(* Logix 5000 project; controller SX_V040001_C001 vendor 1 type 14 code 77 rev 16.22; software revision 16.04; part 29 of 35 *)
(* tags used below, declared in another part *)
   ALL_KINDS : INT[90];
   DRIVE : INT[32];
   DRIVE_INTERVAL : INT[8];
   EMPTYING : INT[18];
   G_DInput : DINT[3];
   loading : INT[19];
   louvre : INT[11];
   METERING : INT[44];
   NOTDOS : INT[6];
   PARAMETER : INT[501];
   pointer_recipe_line : DINT;
   REC_NR_BCD_REMOTE : INT[5];
   REC_NR_BCD_STRING : SINT[2];
   RECIPE_GENERAL : INT[405];
   RM_CMD : INT[9];
   TEMP : INT[14];
(* MainProgram, continued *)

ROUTINE RecipeEnd   (* ladder *)
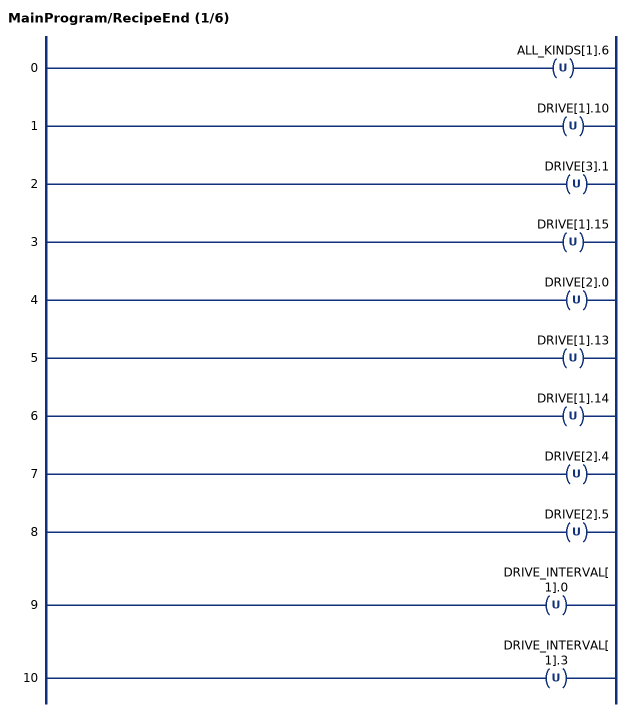
   0: OTU(ALL_KINDS[1].6);
   1: OTU(DRIVE[1].10);
   2: OTU(DRIVE[3].1);
   3: OTU(DRIVE[1].15);
   4: OTU(DRIVE[2].0);
   5: OTU(DRIVE[1].13);
   6: OTU(DRIVE[1].14);
   7: OTU(DRIVE[2].4);
   8: OTU(DRIVE[2].5);
   9: OTU(DRIVE_INTERVAL[1].0);
   10: OTU(DRIVE_INTERVAL[1].3);
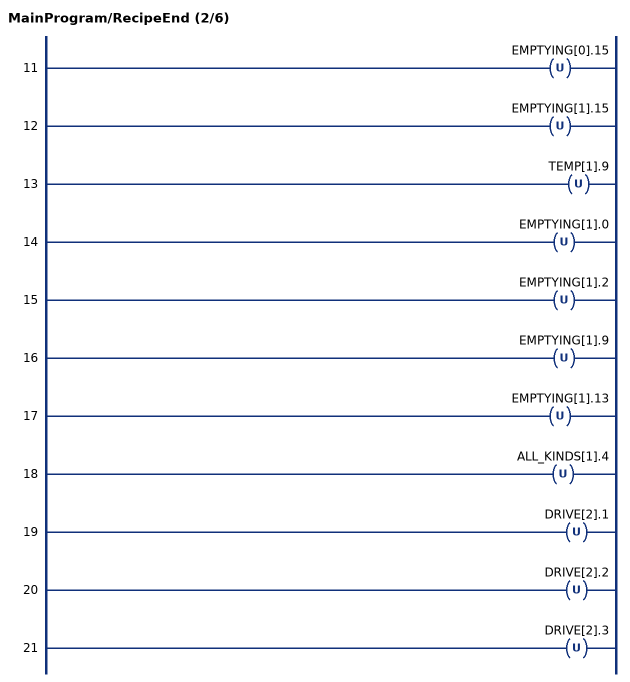
   11: OTU(EMPTYING[0].15);
   12: OTU(EMPTYING[1].15);
   13: OTU(TEMP[1].9);
   14: OTU(EMPTYING[1].0);
   15: OTU(EMPTYING[1].2);
   16: OTU(EMPTYING[1].9);
   17: OTU(EMPTYING[1].13);
   18: OTU(ALL_KINDS[1].4);
   19: OTU(DRIVE[2].1);
   20: OTU(DRIVE[2].2);
   21: OTU(DRIVE[2].3);
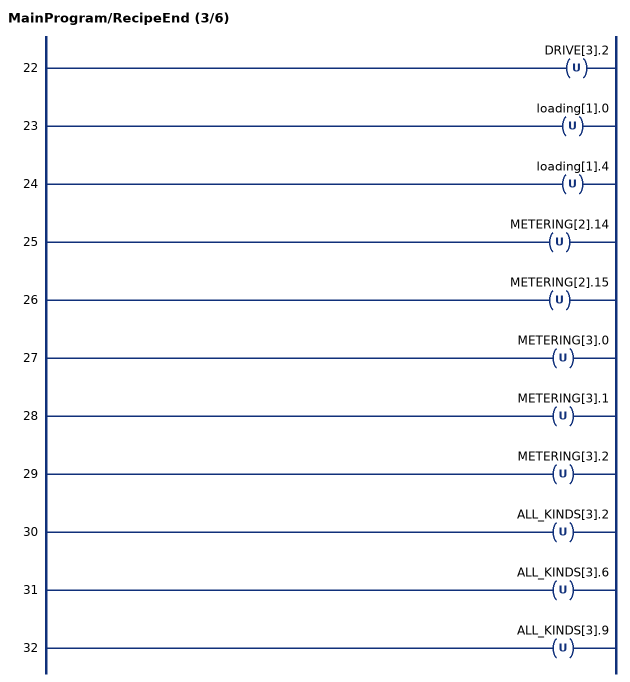
   22: OTU(DRIVE[3].2);
   23: OTU(loading[1].0);
   24: OTU(loading[1].4);
   25: OTU(METERING[2].14);
   26: OTU(METERING[2].15);
   27: OTU(METERING[3].0);
   28: OTU(METERING[3].1);
   29: OTU(METERING[3].2);
   30: OTU(ALL_KINDS[3].2);
   31: OTU(ALL_KINDS[3].6);
   32: OTU(ALL_KINDS[3].9);
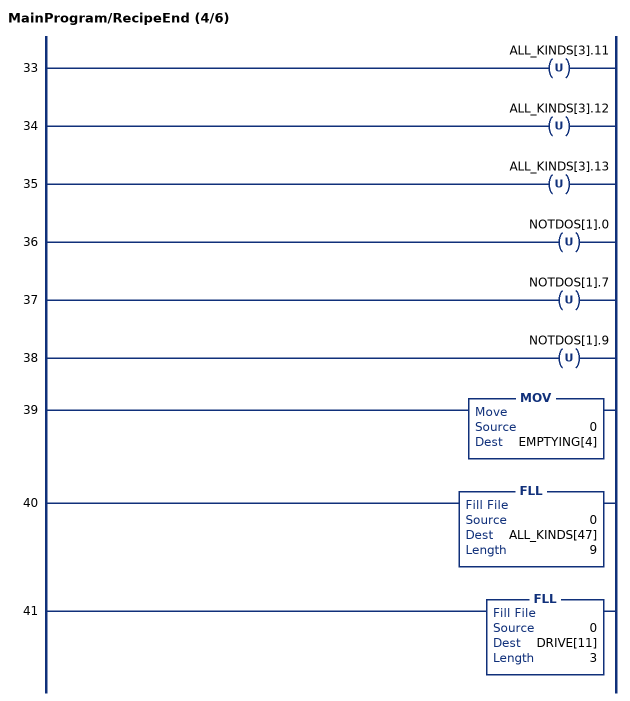
   33: OTU(ALL_KINDS[3].11);
   34: OTU(ALL_KINDS[3].12);
   35: OTU(ALL_KINDS[3].13);
   36: OTU(NOTDOS[1].0);
   37: OTU(NOTDOS[1].7);
   38: OTU(NOTDOS[1].9);
   39: MOV(0,EMPTYING[4]);
   40: FLL(0,ALL_KINDS[47],9);
   41: FLL(0,DRIVE[11],3);
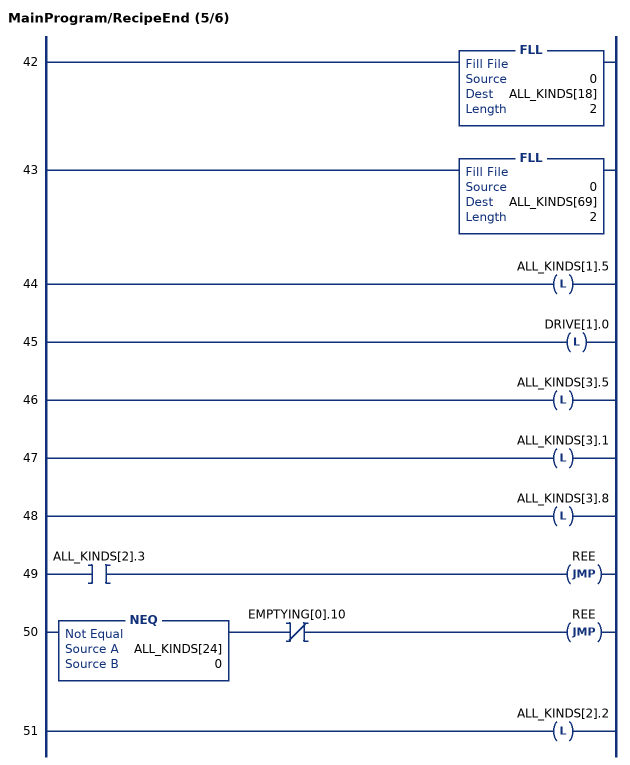
   42: FLL(0,ALL_KINDS[18],2);
   43: FLL(0,ALL_KINDS[69],2);
   44: OTL(ALL_KINDS[1].5);
   45: OTL(DRIVE[1].0);
   46: OTL(ALL_KINDS[3].5);
   47: OTL(ALL_KINDS[3].1);
   48: OTL(ALL_KINDS[3].8);
   49: XIC(ALL_KINDS[2].3)JMP(REE);
   50: NEQ(ALL_KINDS[24],0)XIO(EMPTYING[0].10)JMP(REE);
   51: OTL(ALL_KINDS[2].2);
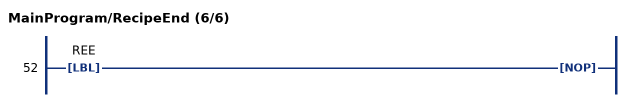
   52: LBL(REE)NOP();
END_ROUTINE

ROUTINE RecipeInterruption   (* ladder *)
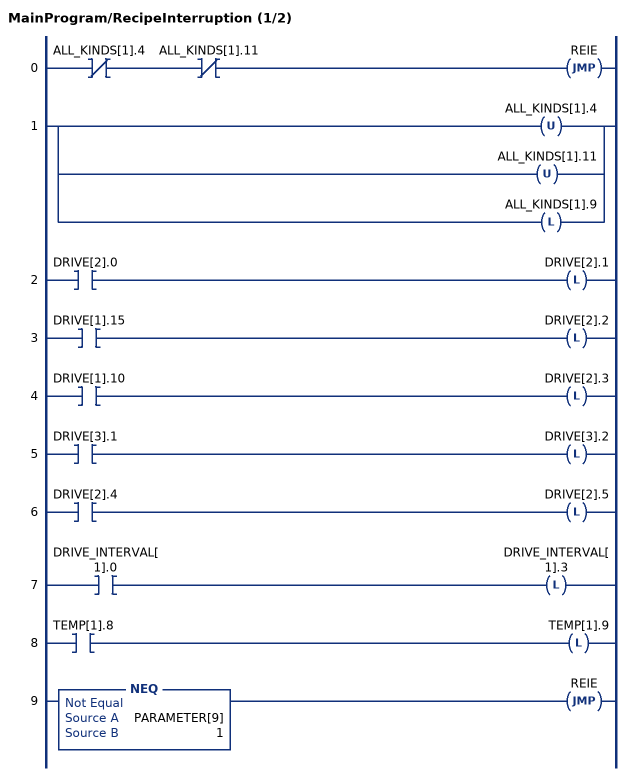
   0: XIO(ALL_KINDS[1].4)XIO(ALL_KINDS[1].11)JMP(REIE);
   1: [OTU(ALL_KINDS[1].4) ,OTU(ALL_KINDS[1].11) ,OTL(ALL_KINDS[1].9) ];
   2: XIC(DRIVE[2].0)OTL(DRIVE[2].1);
   3: XIC(DRIVE[1].15)OTL(DRIVE[2].2);
   4: XIC(DRIVE[1].10)OTL(DRIVE[2].3);
   5: XIC(DRIVE[3].1)OTL(DRIVE[3].2);
   6: XIC(DRIVE[2].4)OTL(DRIVE[2].5);
   7: XIC(DRIVE_INTERVAL[1].0)OTL(DRIVE_INTERVAL[1].3);
   8: XIC(TEMP[1].8)OTL(TEMP[1].9);
   9: NEQ(PARAMETER[9],1)JMP(REIE);
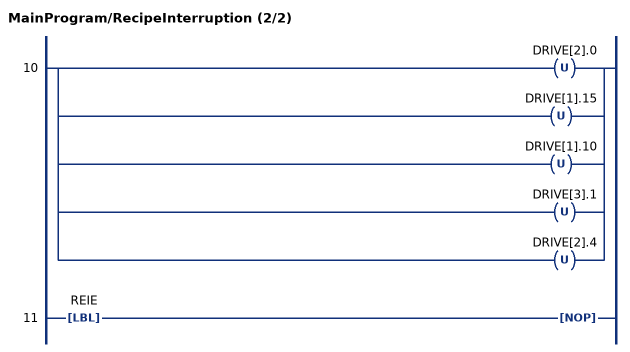
   10: [OTU(DRIVE[2].0) ,OTU(DRIVE[1].15) ,OTU(DRIVE[1].10) ,OTU(DRIVE[3].1) ,OTU(DRIVE[2].4) ];
   11: LBL(REIE)NOP();
END_ROUTINE

ROUTINE RecipeNewstart   (* ladder *)
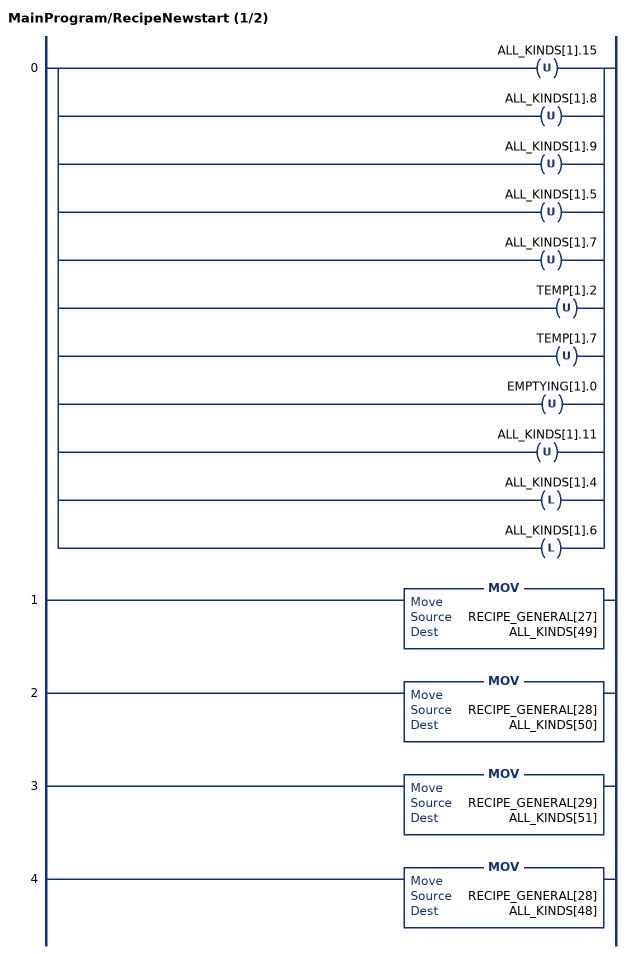
   0: [OTU(ALL_KINDS[1].15) ,OTU(ALL_KINDS[1].8) ,OTU(ALL_KINDS[1].9) ,OTU(ALL_KINDS[1].5) ,OTU(ALL_KINDS[1].7) ,OTU(TEMP[1].2) ,OTU(TEMP[1].7) ,OTU(EMPTYING[1].0) ,OTU(ALL_KINDS[1].11) ,OTL(ALL_KINDS[1].4) ,OTL(ALL_KINDS[1].6) ];
   1: MOV(RECIPE_GENERAL[27],ALL_KINDS[49]);
   2: MOV(RECIPE_GENERAL[28],ALL_KINDS[50]);
   3: MOV(RECIPE_GENERAL[29],ALL_KINDS[51]);
   4: MOV(RECIPE_GENERAL[28],ALL_KINDS[48]);
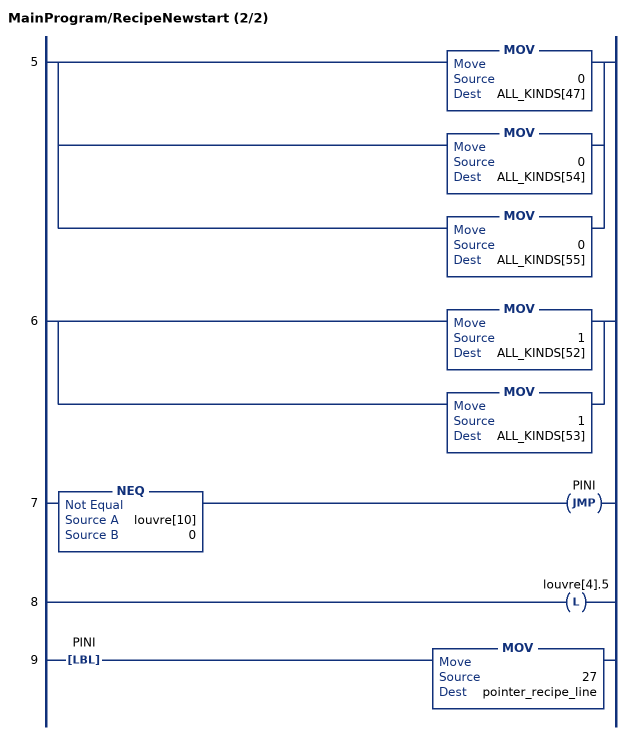
   5: [MOV(0,ALL_KINDS[47]) ,MOV(0,ALL_KINDS[54]) ,MOV(0,ALL_KINDS[55]) ];
   6: [MOV(1,ALL_KINDS[52]) ,MOV(1,ALL_KINDS[53]) ];
   7: NEQ(louvre[10],0)JMP(PINI);
   8: OTL(louvre[4].5);
   9: LBL(PINI)MOV(27,pointer_recipe_line);
END_ROUTINE

ROUTINE RecipeNrBCDin   (* ladder *)
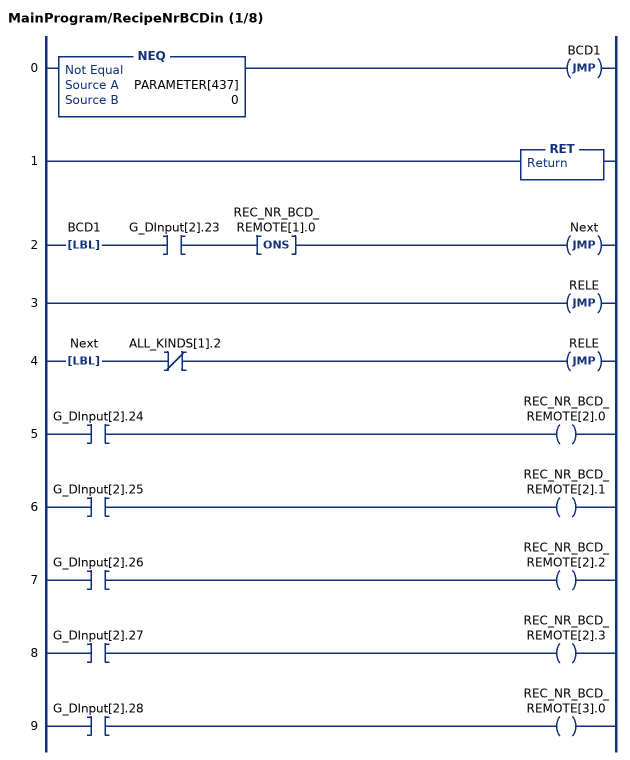
   0: NEQ(PARAMETER[437],0)JMP(BCD1);
   1: RET();
   2: LBL(BCD1)XIC(G_DInput[2].23)ONS(REC_NR_BCD_REMOTE[1].0)JMP(Next);
   3: JMP(RELE);
   4: LBL(Next)XIO(ALL_KINDS[1].2)JMP(RELE);
   5: XIC(G_DInput[2].24)OTE(REC_NR_BCD_REMOTE[2].0);
   6: XIC(G_DInput[2].25)OTE(REC_NR_BCD_REMOTE[2].1);
   7: XIC(G_DInput[2].26)OTE(REC_NR_BCD_REMOTE[2].2);
   8: XIC(G_DInput[2].27)OTE(REC_NR_BCD_REMOTE[2].3);
   9: XIC(G_DInput[2].28)OTE(REC_NR_BCD_REMOTE[3].0);
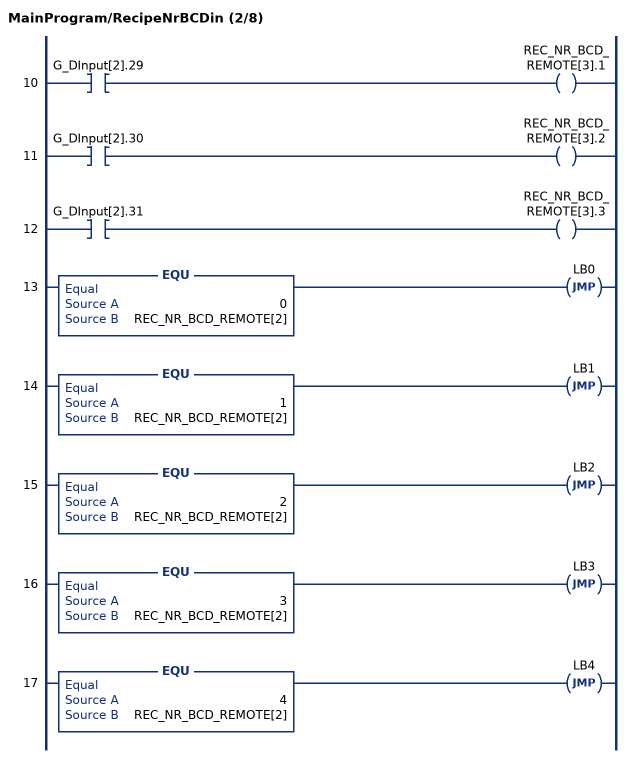
   10: XIC(G_DInput[2].29)OTE(REC_NR_BCD_REMOTE[3].1);
   11: XIC(G_DInput[2].30)OTE(REC_NR_BCD_REMOTE[3].2);
   12: XIC(G_DInput[2].31)OTE(REC_NR_BCD_REMOTE[3].3);
   13: EQU(0,REC_NR_BCD_REMOTE[2])JMP(LB0);
   14: EQU(1,REC_NR_BCD_REMOTE[2])JMP(LB1);
   15: EQU(2,REC_NR_BCD_REMOTE[2])JMP(LB2);
   16: EQU(3,REC_NR_BCD_REMOTE[2])JMP(LB3);
   17: EQU(4,REC_NR_BCD_REMOTE[2])JMP(LB4);
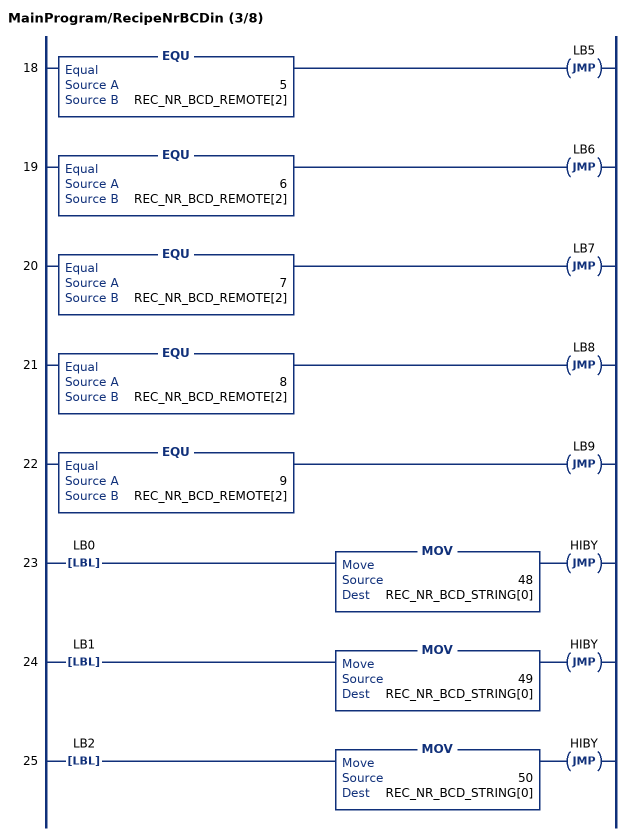
   18: EQU(5,REC_NR_BCD_REMOTE[2])JMP(LB5);
   19: EQU(6,REC_NR_BCD_REMOTE[2])JMP(LB6);
   20: EQU(7,REC_NR_BCD_REMOTE[2])JMP(LB7);
   21: EQU(8,REC_NR_BCD_REMOTE[2])JMP(LB8);
   22: EQU(9,REC_NR_BCD_REMOTE[2])JMP(LB9);
   23: LBL(LB0)MOV(48,REC_NR_BCD_STRING[0])JMP(HIBY);
   24: LBL(LB1)MOV(49,REC_NR_BCD_STRING[0])JMP(HIBY);
   25: LBL(LB2)MOV(50,REC_NR_BCD_STRING[0])JMP(HIBY);
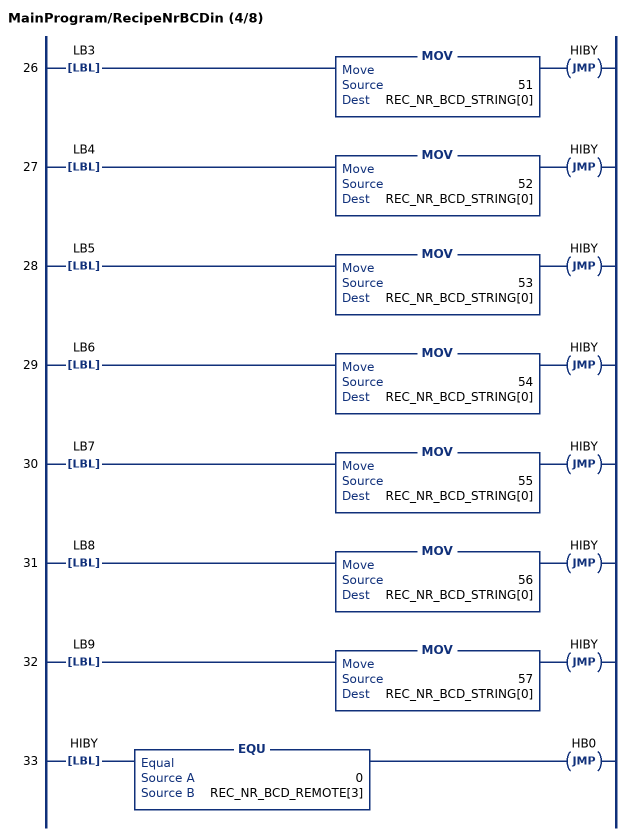
   26: LBL(LB3)MOV(51,REC_NR_BCD_STRING[0])JMP(HIBY);
   27: LBL(LB4)MOV(52,REC_NR_BCD_STRING[0])JMP(HIBY);
   28: LBL(LB5)MOV(53,REC_NR_BCD_STRING[0])JMP(HIBY);
   29: LBL(LB6)MOV(54,REC_NR_BCD_STRING[0])JMP(HIBY);
   30: LBL(LB7)MOV(55,REC_NR_BCD_STRING[0])JMP(HIBY);
   31: LBL(LB8)MOV(56,REC_NR_BCD_STRING[0])JMP(HIBY);
   32: LBL(LB9)MOV(57,REC_NR_BCD_STRING[0])JMP(HIBY);
   33: LBL(HIBY)EQU(0,REC_NR_BCD_REMOTE[3])JMP(HB0);
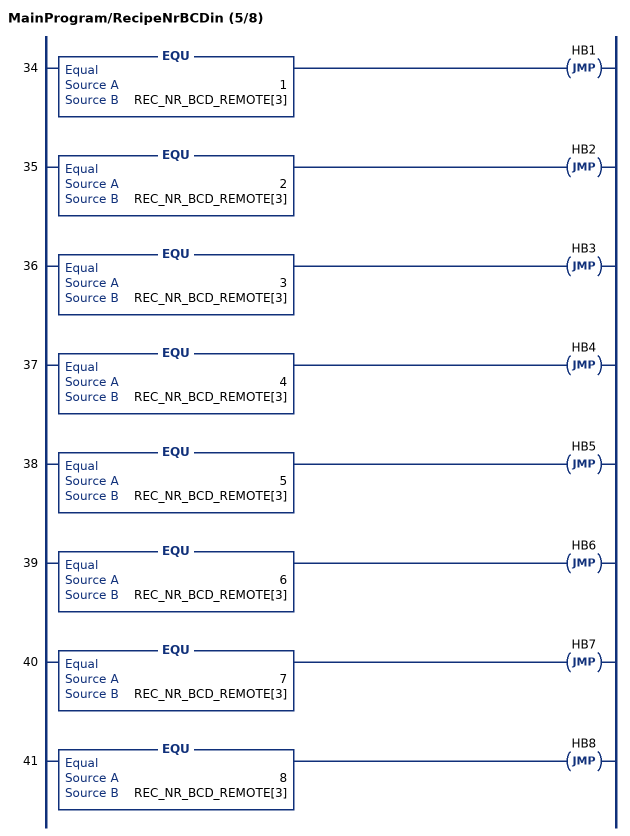
   34: EQU(1,REC_NR_BCD_REMOTE[3])JMP(HB1);
   35: EQU(2,REC_NR_BCD_REMOTE[3])JMP(HB2);
   36: EQU(3,REC_NR_BCD_REMOTE[3])JMP(HB3);
   37: EQU(4,REC_NR_BCD_REMOTE[3])JMP(HB4);
   38: EQU(5,REC_NR_BCD_REMOTE[3])JMP(HB5);
   39: EQU(6,REC_NR_BCD_REMOTE[3])JMP(HB6);
   40: EQU(7,REC_NR_BCD_REMOTE[3])JMP(HB7);
   41: EQU(8,REC_NR_BCD_REMOTE[3])JMP(HB8);
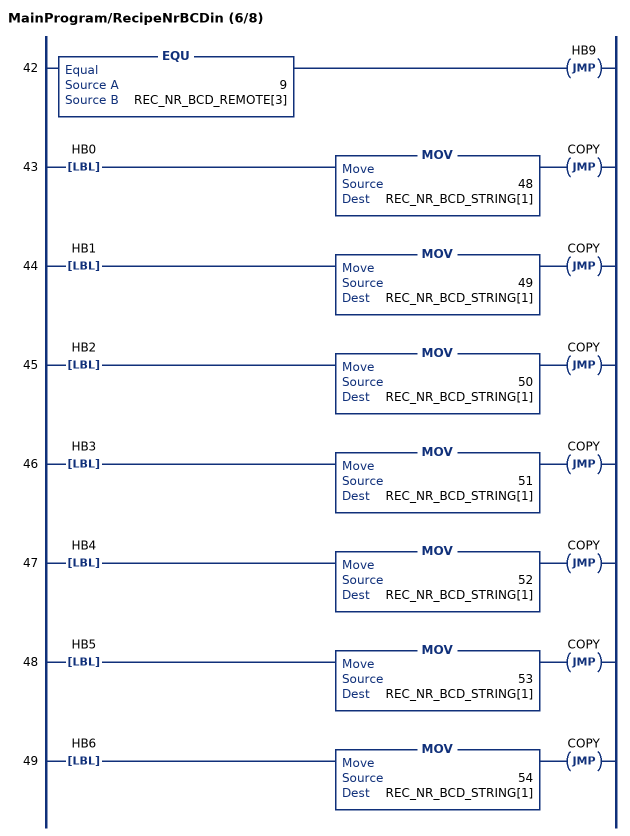
   42: EQU(9,REC_NR_BCD_REMOTE[3])JMP(HB9);
   43: LBL(HB0)MOV(48,REC_NR_BCD_STRING[1])JMP(COPY);
   44: LBL(HB1)MOV(49,REC_NR_BCD_STRING[1])JMP(COPY);
   45: LBL(HB2)MOV(50,REC_NR_BCD_STRING[1])JMP(COPY);
   46: LBL(HB3)MOV(51,REC_NR_BCD_STRING[1])JMP(COPY);
   47: LBL(HB4)MOV(52,REC_NR_BCD_STRING[1])JMP(COPY);
   48: LBL(HB5)MOV(53,REC_NR_BCD_STRING[1])JMP(COPY);
   49: LBL(HB6)MOV(54,REC_NR_BCD_STRING[1])JMP(COPY);
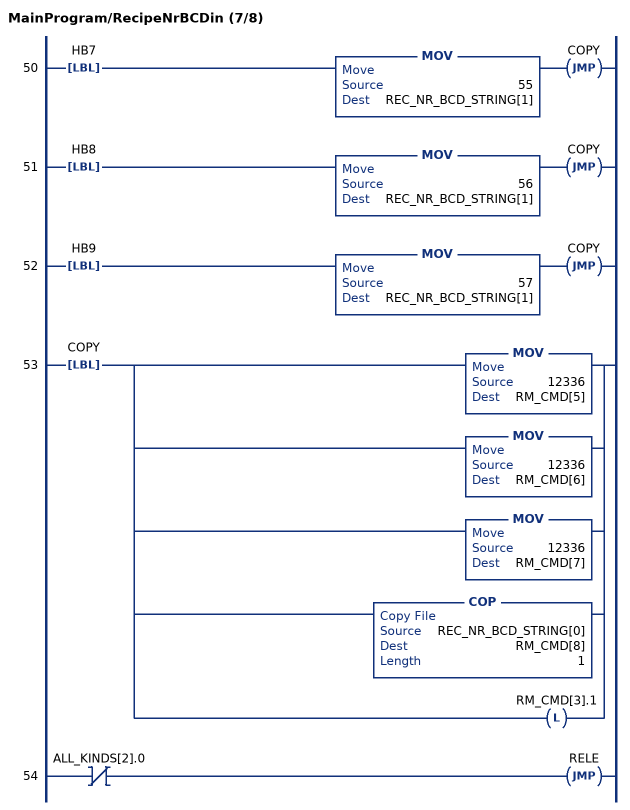
   50: LBL(HB7)MOV(55,REC_NR_BCD_STRING[1])JMP(COPY);
   51: LBL(HB8)MOV(56,REC_NR_BCD_STRING[1])JMP(COPY);
   52: LBL(HB9)MOV(57,REC_NR_BCD_STRING[1])JMP(COPY);
   53: LBL(COPY)[MOV(12336,RM_CMD[5]) ,MOV(12336,RM_CMD[6]) ,MOV(12336,RM_CMD[7]) ,COP(REC_NR_BCD_STRING[0],RM_CMD[8],1) ,OTL(RM_CMD[3].1) ];
   54: XIO(ALL_KINDS[2].0)JMP(RELE);
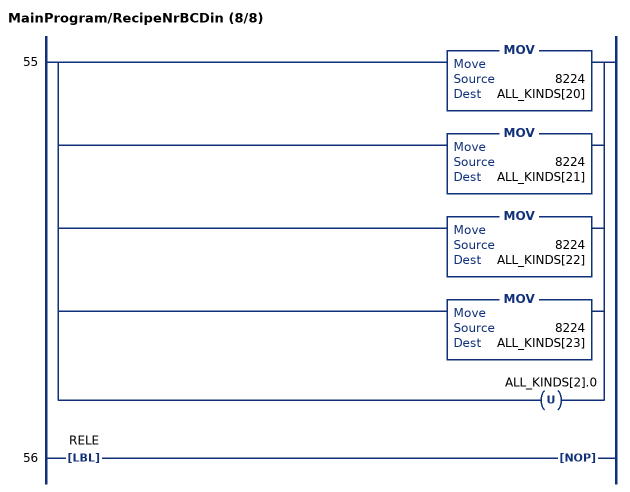
   55: [MOV(8224,ALL_KINDS[20]) ,MOV(8224,ALL_KINDS[21]) ,MOV(8224,ALL_KINDS[22]) ,MOV(8224,ALL_KINDS[23]) ,OTU(ALL_KINDS[2].0) ];
   56: LBL(RELE)NOP();
END_ROUTINE
